(* Schneider Machine Expert - Basic project es3_4pompe_3max_4soglie_misura_livello_con_alternanza_semplice_a_livello_minimo, file version 3.0.0.0 *)
(* ProjectInformations: Name=New project *)

HARDWARE
  Cpu 0: TM221C40R
  ModuleExtensionObject 0: TM3AI8/G
  EthernetConfiguration: NetworkName=M221, IpAllocationMode=FixedAddress, IpAddress=0.0.0.0, SubnetMask=0.0.0.0
  SerialLineConfiguration: Baud=Baud19200, Parity=ParityEven, DataBits=DataBits8, StopBits=StopBits1, PhysicalMedium=PhysicalMediumRs485, TransmissionMode=TransmissionModeModbusRtu, SlaveId=1, Addressing=SlaveAddressing
  MastTask: UsePeriodScanMode=false, PeriodScan=100
  FastTask: Period=255
  CpuBehavior: StartingMode=StartAsPreviousState, AutoSaveRamOnEeprom=true, WatchdogPeriod=250

SYMBOLS  (address, symbol, comment, settings)
  %M0       P1_USABILE
  %M1       P2_USABILE
  %M2       SOTTO_SOGLIA_MIN  "Il livello acqua è passato sotto la soglia minima?"
  %M3       SOPRA_SOGLIA_MAX1  "Il livello acqua è passato sopra la soglia 1 massima?"
  %M4       SOPRA_SOGLIA_MAX2  "Il livello acqua è passato sopra la soglia 2 massima?"
  %M5       PASSATO_SOGLIA_MAX3
  %M6       P1_COMANDATA
  %M7       P2_COMANDATA
  %M8       P3_USABILE
  %M9       P4_USABILE
  %M10      P3_COMANDATA
  %M11      P4_COMANDATA
  %M12      SOPRA_SOGLIA_MAX3  "Il livello acqua è passato sopra la soglia 3 massima?"
  %M13      PASSATO_SOGLIA_MAX2
  %M14      PASSATO_SOGLIA_MAX1
  %MW0      LVL_PERC  "Livello acqua percentuale."
  %MW1      NUM_POMPE_DA_COMANDARE
  %MW2      NUM_POMPE_COMANDATE
  %MD1      LVL_CALC_TMP
  %KD0      MIN_SCALA_GREZZO  [Value=1310724000]
  %KD1      MAX_SCALA_GREZZO  [Value=20000]
  %I0.0     P1_AUTO
  %I0.1     P1_MOTO
  %I0.2     P1_ANOMALIA
  %I0.3     P2_AUTO
  %I0.4     P2_MOTO
  %I0.5     P2_ANOMALIA
  %I0.6     P3_AUTO
  %I0.7     P3_MOTO
  %I0.8     P3_ANOMALIA
  %I0.9     P4_AUTO
  %I0.10    P4_MOTO
  %I0.11    P4_ANOMALIA
  %Q0.0     P1_CMD
  %Q0.1     P2_CMD
  %Q0.2     P3_CMD
  %Q0.3     P4_CMD
  %IW1.0    LVL_INPUT_GREZZO  [Type=Type_4_20mA, Scope=Scope_Customized, Minimum=4000, Maximum=20000]
  %IW1.1    SOGLIA_MIN_PERC  [Type=Type_0_10V, Scope=Scope_Customized, Minimum=0, Maximum=100]
  %IW1.2    SOGLIA_MAX1_PERC  [Type=Type_0_10V, Scope=Scope_Customized, Minimum=0, Maximum=100]
  %IW1.3    SOGLIA_MAX2_PERC  [Type=Type_0_10V, Scope=Scope_Customized, Minimum=0, Maximum=100]
  %IW1.4    SOGLIA_MAX3_PERC  [Type=Type_0_10V, Scope=Scope_Customized, Minimum=0, Maximum=100]

POU Main
  (* SectionNumber=1 *)

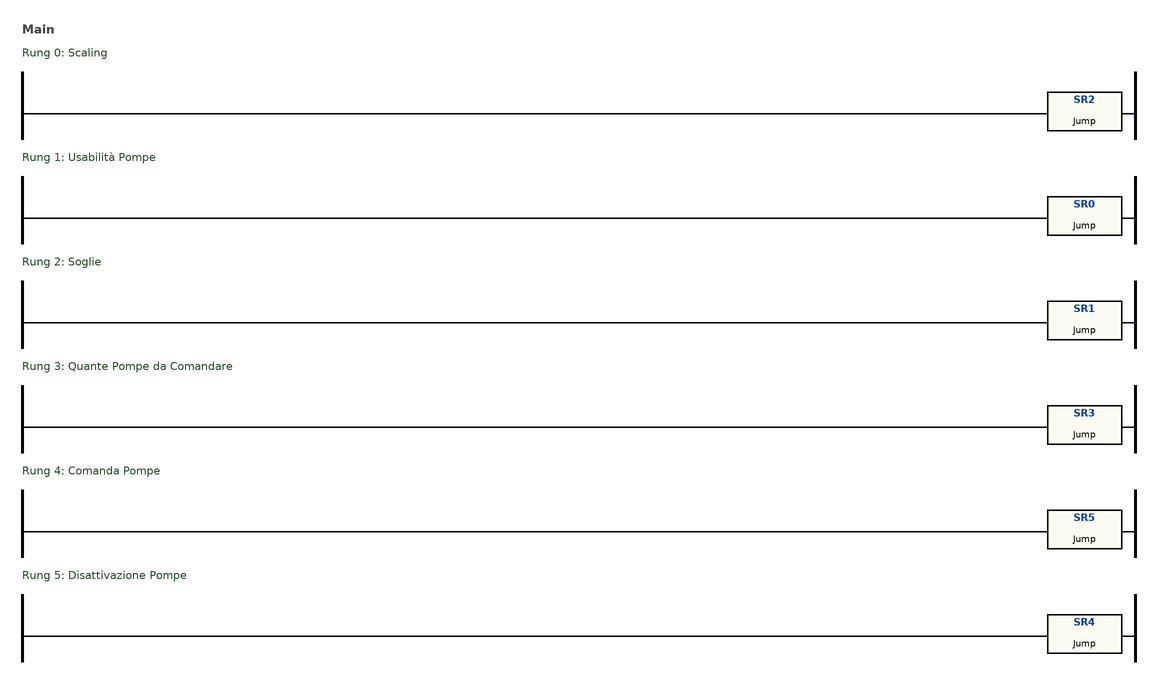

// Rung 0: Scaling
  LD 1
  SR2
  // as ST:
  //   SR2();

// Rung 1: Usabilità Pompe
  LD 1
  SR0
  // as ST:
  //   SR0();

// Rung 2: Soglie
  LD 1
  SR1
  // as ST:
  //   SR1();

// Rung 3: Quante Pompe da Comandare
  LD 1
  SR3
  // as ST:
  //   SR3();

// Rung 4: Comanda Pompe
  LD 1
  SR5
  // as ST:
  //   SR5();

// Rung 5: Disattivazione Pompe
  LD 1
  SR4
  // as ST:
  //   SR4();

Subroutine Usabilità Pompe
  (* SectionNumber=2, Number=0 *)

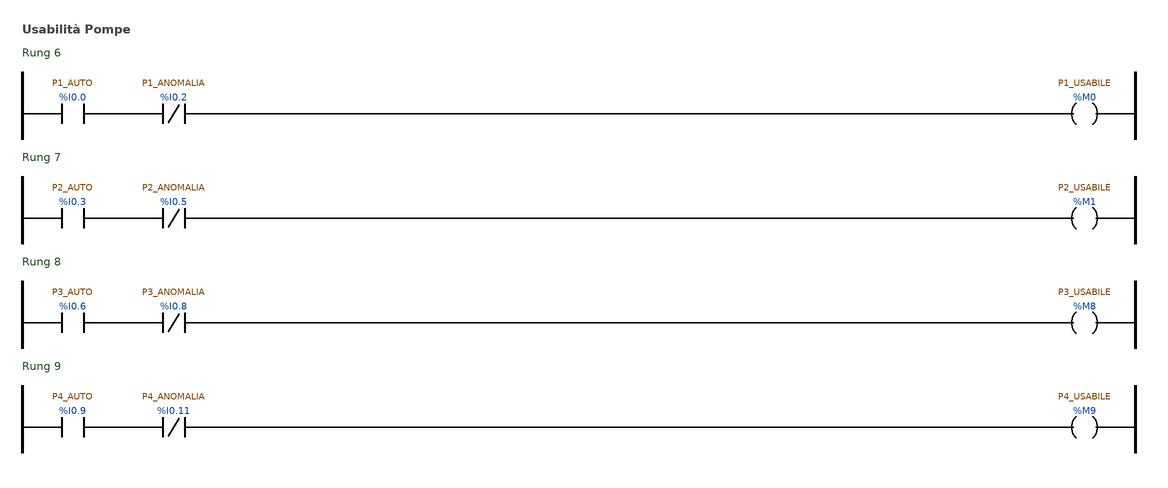

// Rung 6
  LD %I0.0                (* P1_AUTO *)
  ANDN %I0.2              (* P1_ANOMALIA *)
  ST %M0                  (* P1_USABILE *)
  // as ST:
  //   P1_USABILE := P1_AUTO AND NOT P1_ANOMALIA;

// Rung 7
  LD %I0.3                (* P2_AUTO *)
  ANDN %I0.5              (* P2_ANOMALIA *)
  ST %M1                  (* P2_USABILE *)
  // as ST:
  //   P2_USABILE := P2_AUTO AND NOT P2_ANOMALIA;

// Rung 8
  LD %I0.6                (* P3_AUTO *)
  ANDN %I0.8              (* P3_ANOMALIA *)
  ST %M8                  (* P3_USABILE *)
  // as ST:
  //   P3_USABILE := P3_AUTO AND NOT P3_ANOMALIA;

// Rung 9
  LD %I0.9                (* P4_AUTO *)
  ANDN %I0.11             (* P4_ANOMALIA *)
  ST %M9                  (* P4_USABILE *)
  // as ST:
  //   P4_USABILE := P4_AUTO AND NOT P4_ANOMALIA;

Subroutine Soglie
  (* SectionNumber=3, Number=1 *)

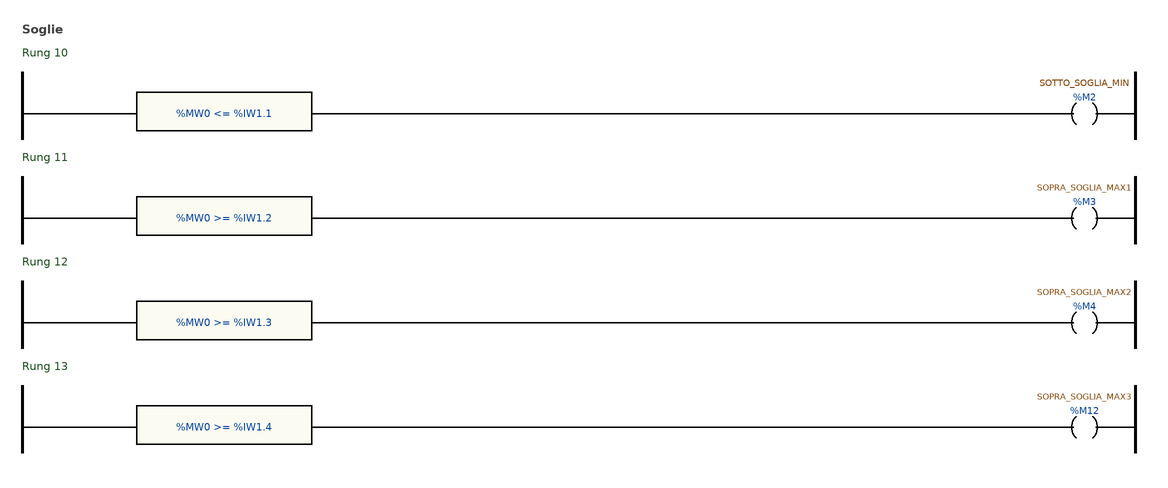

// Rung 10
  LD [ %MW0 <= %IW1.1 ]   (* LVL_PERC, SOGLIA_MIN_PERC *)
  ST %M2                  (* SOTTO_SOGLIA_MIN *)
  // as ST:
  //   SOTTO_SOGLIA_MIN := LVL_PERC <= SOGLIA_MIN_PERC;

// Rung 11
  LD [ %MW0 >= %IW1.2 ]   (* LVL_PERC, SOGLIA_MAX1_PERC *)
  ST %M3                  (* SOPRA_SOGLIA_MAX1 *)
  // as ST:
  //   SOPRA_SOGLIA_MAX1 := LVL_PERC >= SOGLIA_MAX1_PERC;

// Rung 12
  LD [ %MW0 >= %IW1.3 ]   (* LVL_PERC, SOGLIA_MAX2_PERC *)
  ST %M4                  (* SOPRA_SOGLIA_MAX2 *)
  // as ST:
  //   SOPRA_SOGLIA_MAX2 := LVL_PERC >= SOGLIA_MAX2_PERC;

// Rung 13
  LD [ %MW0 >= %IW1.4 ]   (* LVL_PERC, SOGLIA_MAX3_PERC *)
  ST %M12                 (* SOPRA_SOGLIA_MAX3 *)
  // as ST:
  //   SOPRA_SOGLIA_MAX3 := LVL_PERC >= SOGLIA_MAX3_PERC;

Subroutine Scaling
  (* SectionNumber=4, Number=2 *)

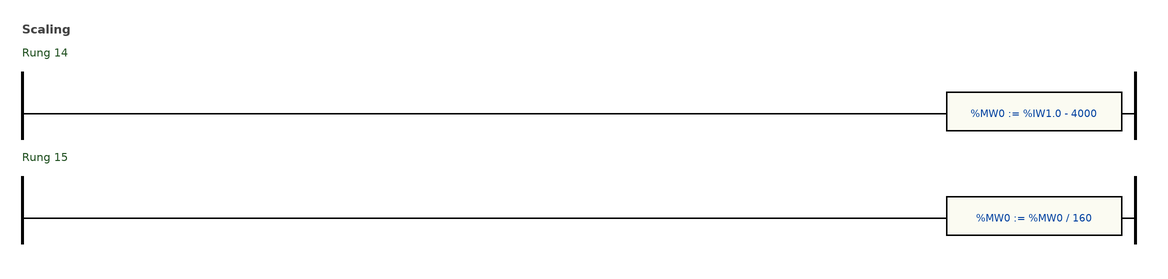

// Rung 14
  LD 1
  [ %MW0 := %IW1.0 - 4000 ](* LVL_PERC, LVL_INPUT_GREZZO *)
  // as ST:
  //   LVL_PERC := LVL_INPUT_GREZZO - 4000;

// Rung 15
  LD 1
  [ %MW0 := %MW0 / 160 ]  (* LVL_PERC, LVL_PERC *)
  // as ST:
  //   LVL_PERC := LVL_PERC / 160;

Subroutine Quante Pompe da Comandare
  (* SectionNumber=5, Number=3 *)

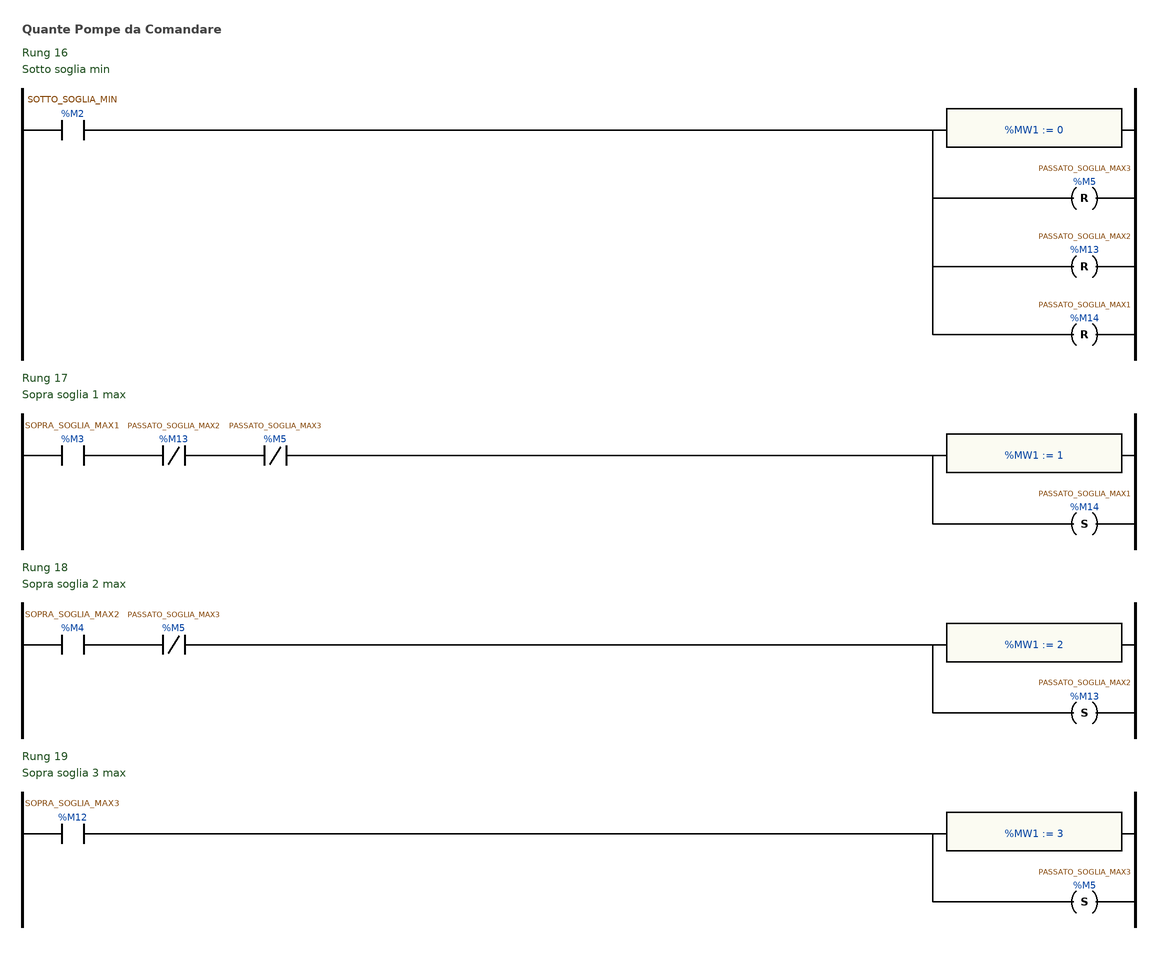

// Rung 16
// Sotto soglia min
  LD %M2                  (* SOTTO_SOGLIA_MIN *)
  [ %MW1 := 0 ]           (* NUM_POMPE_DA_COMANDARE *)
  R %M5                   (* PASSATO_SOGLIA_MAX3 *)
  R %M13                  (* PASSATO_SOGLIA_MAX2 *)
  R %M14                  (* PASSATO_SOGLIA_MAX1 *)
  // as ST:
  //   IF SOTTO_SOGLIA_MIN THEN NUM_POMPE_DA_COMANDARE := 0; END_IF;
  //   IF SOTTO_SOGLIA_MIN THEN PASSATO_SOGLIA_MAX3 := FALSE; END_IF;
  //   IF SOTTO_SOGLIA_MIN THEN PASSATO_SOGLIA_MAX2 := FALSE; END_IF;
  //   IF SOTTO_SOGLIA_MIN THEN PASSATO_SOGLIA_MAX1 := FALSE; END_IF;

// Rung 17
// Sopra soglia 1 max
  LD %M3                  (* SOPRA_SOGLIA_MAX1 *)
  ANDN %M13               (* PASSATO_SOGLIA_MAX2 *)
  ANDN %M5                (* PASSATO_SOGLIA_MAX3 *)
  [ %MW1 := 1 ]           (* NUM_POMPE_DA_COMANDARE *)
  S %M14                  (* PASSATO_SOGLIA_MAX1 *)
  // as ST:
  //   IF SOPRA_SOGLIA_MAX1 AND NOT PASSATO_SOGLIA_MAX2 AND NOT PASSATO_SOGLIA_MAX3 THEN NUM_POMPE_DA_COMANDARE := 1; END_IF;
  //   IF SOPRA_SOGLIA_MAX1 AND NOT PASSATO_SOGLIA_MAX2 AND NOT PASSATO_SOGLIA_MAX3 THEN PASSATO_SOGLIA_MAX1 := TRUE; END_IF;

// Rung 18
// Sopra soglia 2 max
  LD %M4                  (* SOPRA_SOGLIA_MAX2 *)
  ANDN %M5                (* PASSATO_SOGLIA_MAX3 *)
  [ %MW1 := 2 ]           (* NUM_POMPE_DA_COMANDARE *)
  S %M13                  (* PASSATO_SOGLIA_MAX2 *)
  // as ST:
  //   IF SOPRA_SOGLIA_MAX2 AND NOT PASSATO_SOGLIA_MAX3 THEN NUM_POMPE_DA_COMANDARE := 2; END_IF;
  //   IF SOPRA_SOGLIA_MAX2 AND NOT PASSATO_SOGLIA_MAX3 THEN PASSATO_SOGLIA_MAX2 := TRUE; END_IF;

// Rung 19
// Sopra soglia 3 max
  LD %M12                 (* SOPRA_SOGLIA_MAX3 *)
  [ %MW1 := 3 ]           (* NUM_POMPE_DA_COMANDARE *)
  S %M5                   (* PASSATO_SOGLIA_MAX3 *)
  // as ST:
  //   IF SOPRA_SOGLIA_MAX3 THEN NUM_POMPE_DA_COMANDARE := 3; END_IF;
  //   IF SOPRA_SOGLIA_MAX3 THEN PASSATO_SOGLIA_MAX3 := TRUE; END_IF;

Subroutine Disattivazione Pompe
  (* SectionNumber=6, Number=4 *)

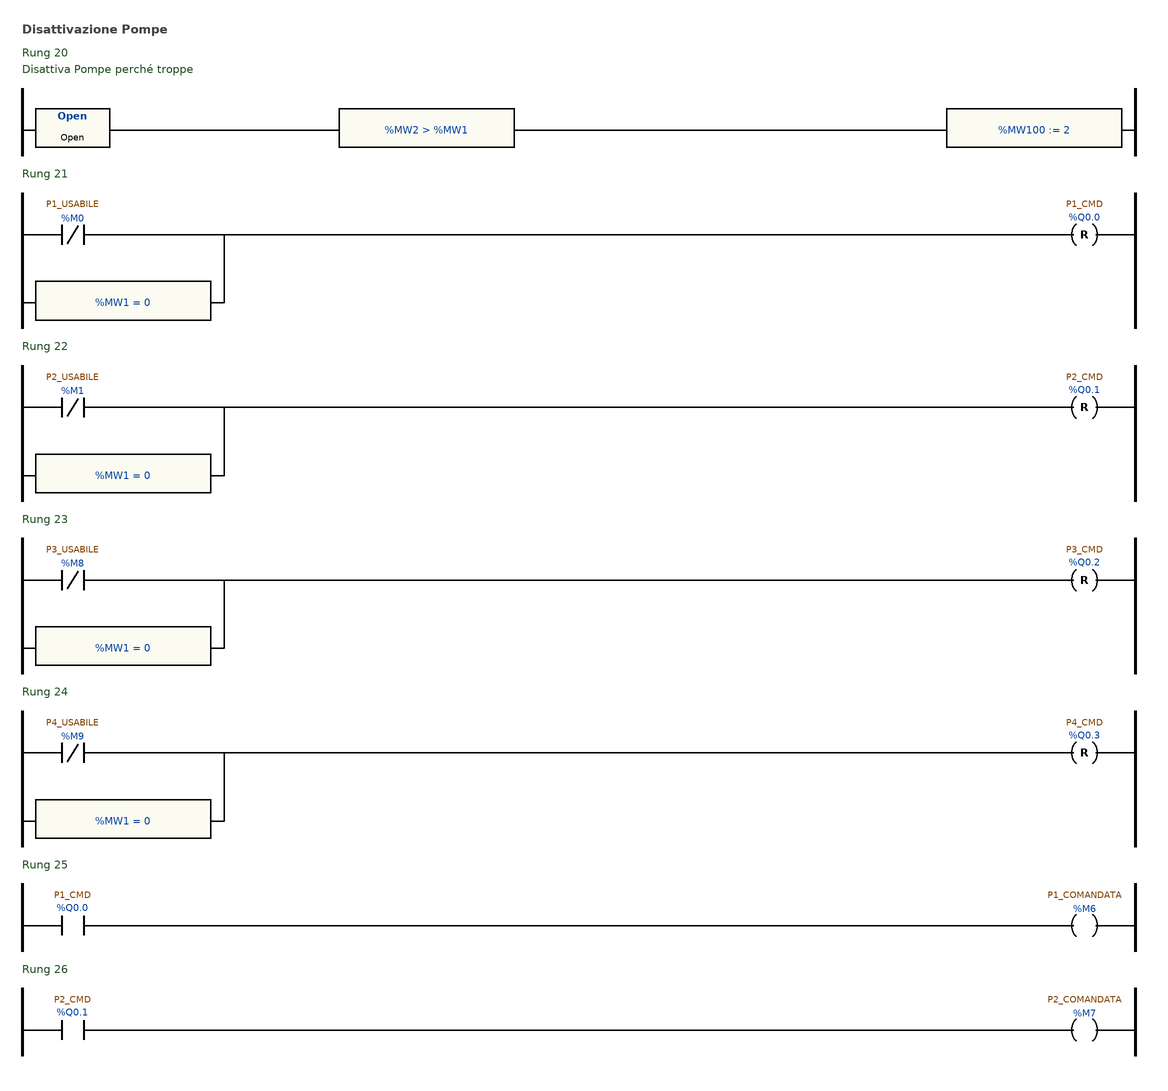

// Rung 20
// Disattiva Pompe perché troppe
  LD 0
  AND [ %MW2 > %MW1 ]     (* NUM_POMPE_COMANDATE, NUM_POMPE_DA_COMANDARE *)
  [ %MW100 := 2 ]
  // as ST:
  //   IF FALSE AND NUM_POMPE_COMANDATE > NUM_POMPE_DA_COMANDARE THEN %MW100 := 2; END_IF;

// Rung 21
  LDN %M0                 (* P1_USABILE *)
  OR [ %MW1 = 0 ]         (* NUM_POMPE_DA_COMANDARE *)
  R %Q0.0                 (* P1_CMD *)
  // as ST:
  //   IF NOT P1_USABILE OR NUM_POMPE_DA_COMANDARE = 0 THEN P1_CMD := FALSE; END_IF;

// Rung 22
  LDN %M1                 (* P2_USABILE *)
  OR [ %MW1 = 0 ]         (* NUM_POMPE_DA_COMANDARE *)
  R %Q0.1                 (* P2_CMD *)
  // as ST:
  //   IF NOT P2_USABILE OR NUM_POMPE_DA_COMANDARE = 0 THEN P2_CMD := FALSE; END_IF;

// Rung 23
  LDN %M8                 (* P3_USABILE *)
  OR [ %MW1 = 0 ]         (* NUM_POMPE_DA_COMANDARE *)
  R %Q0.2                 (* P3_CMD *)
  // as ST:
  //   IF NOT P3_USABILE OR NUM_POMPE_DA_COMANDARE = 0 THEN P3_CMD := FALSE; END_IF;

// Rung 24
  LDN %M9                 (* P4_USABILE *)
  OR [ %MW1 = 0 ]         (* NUM_POMPE_DA_COMANDARE *)
  R %Q0.3                 (* P4_CMD *)
  // as ST:
  //   IF NOT P4_USABILE OR NUM_POMPE_DA_COMANDARE = 0 THEN P4_CMD := FALSE; END_IF;

// Rung 25
  LD %Q0.0                (* P1_CMD *)
  ST %M6                  (* P1_COMANDATA *)
  // as ST:
  //   P1_COMANDATA := P1_CMD;

// Rung 26
  LD %Q0.1                (* P2_CMD *)
  ST %M7                  (* P2_COMANDATA *)
  // as ST:
  //   P2_COMANDATA := P2_CMD;

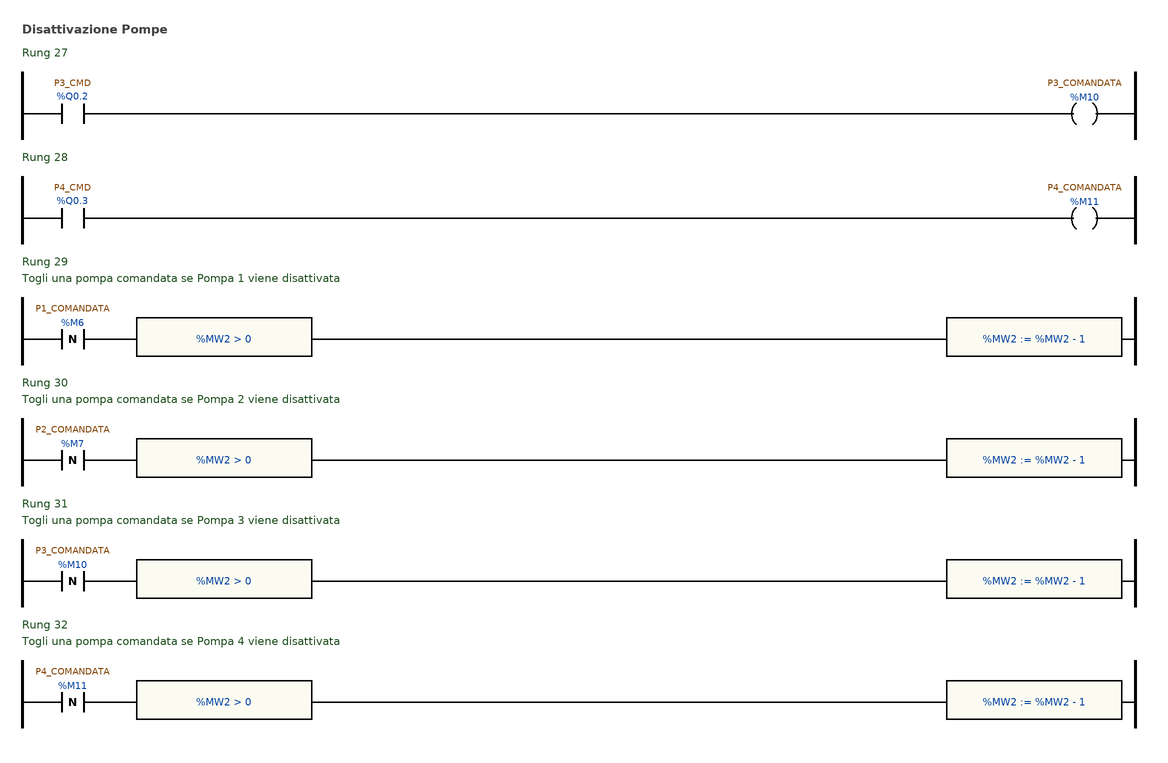

// Rung 27
  LD %Q0.2                (* P3_CMD *)
  ST %M10                 (* P3_COMANDATA *)
  // as ST:
  //   P3_COMANDATA := P3_CMD;

// Rung 28
  LD %Q0.3                (* P4_CMD *)
  ST %M11                 (* P4_COMANDATA *)
  // as ST:
  //   P4_COMANDATA := P4_CMD;

// Rung 29
// Togli una pompa comandata se Pompa 1 viene disattivata
  LDF %M6                 (* P1_COMANDATA *)
  AND [ %MW2 > 0 ]        (* NUM_POMPE_COMANDATE *)
  [ %MW2 := %MW2 - 1 ]    (* NUM_POMPE_COMANDATE, NUM_POMPE_COMANDATE *)
  // as ST:
  //   IF FALLING(P1_COMANDATA) AND NUM_POMPE_COMANDATE > 0 THEN NUM_POMPE_COMANDATE := NUM_POMPE_COMANDATE - 1; END_IF;

// Rung 30
// Togli una pompa comandata se Pompa 2 viene disattivata
  LDF %M7                 (* P2_COMANDATA *)
  AND [ %MW2 > 0 ]        (* NUM_POMPE_COMANDATE *)
  [ %MW2 := %MW2 - 1 ]    (* NUM_POMPE_COMANDATE, NUM_POMPE_COMANDATE *)
  // as ST:
  //   IF FALLING(P2_COMANDATA) AND NUM_POMPE_COMANDATE > 0 THEN NUM_POMPE_COMANDATE := NUM_POMPE_COMANDATE - 1; END_IF;

// Rung 31
// Togli una pompa comandata se Pompa 3 viene disattivata
  LDF %M10                (* P3_COMANDATA *)
  AND [ %MW2 > 0 ]        (* NUM_POMPE_COMANDATE *)
  [ %MW2 := %MW2 - 1 ]    (* NUM_POMPE_COMANDATE, NUM_POMPE_COMANDATE *)
  // as ST:
  //   IF FALLING(P3_COMANDATA) AND NUM_POMPE_COMANDATE > 0 THEN NUM_POMPE_COMANDATE := NUM_POMPE_COMANDATE - 1; END_IF;

// Rung 32
// Togli una pompa comandata se Pompa 4 viene disattivata
  LDF %M11                (* P4_COMANDATA *)
  AND [ %MW2 > 0 ]        (* NUM_POMPE_COMANDATE *)
  [ %MW2 := %MW2 - 1 ]    (* NUM_POMPE_COMANDATE, NUM_POMPE_COMANDATE *)
  // as ST:
  //   IF FALLING(P4_COMANDATA) AND NUM_POMPE_COMANDATE > 0 THEN NUM_POMPE_COMANDATE := NUM_POMPE_COMANDATE - 1; END_IF;

Subroutine Comanda Pompe
  (* SectionNumber=7, Number=5 *)

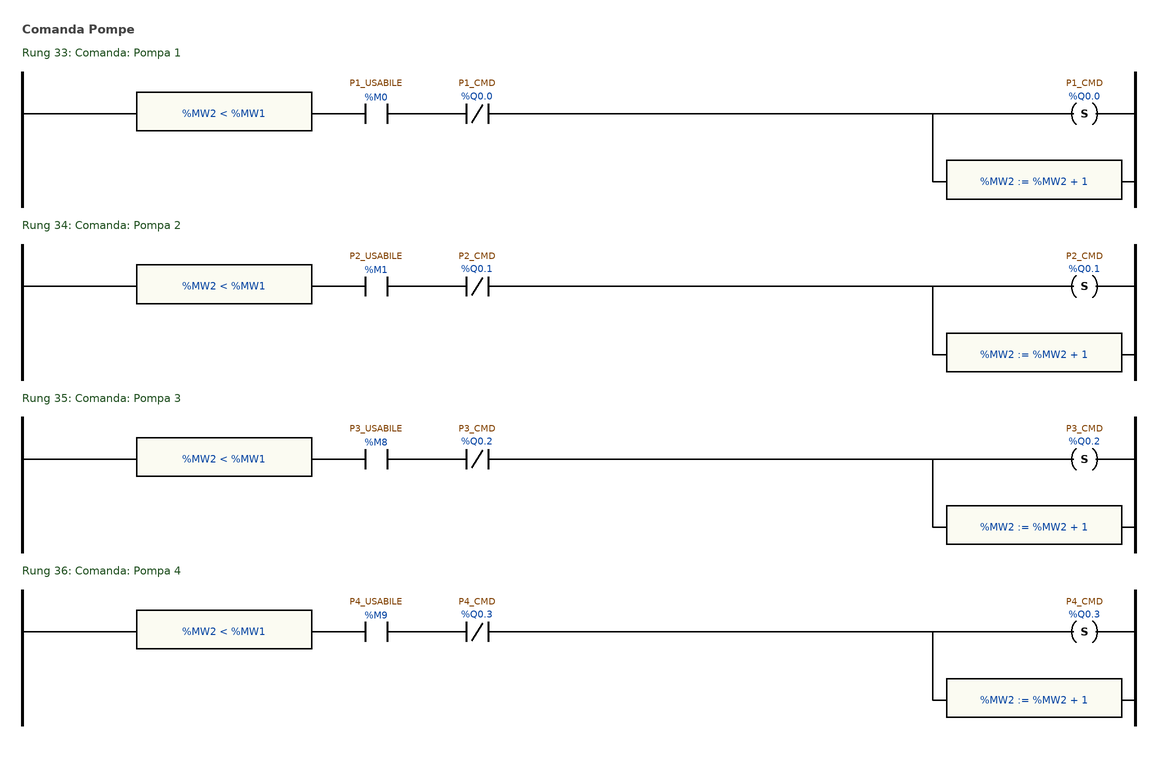

// Rung 33: Comanda: Pompa 1
  LD [ %MW2 < %MW1 ]      (* NUM_POMPE_COMANDATE, NUM_POMPE_DA_COMANDARE *)
  AND %M0                 (* P1_USABILE *)
  ANDN %Q0.0              (* P1_CMD *)
  S %Q0.0                 (* P1_CMD *)
  [ %MW2 := %MW2 + 1 ]    (* NUM_POMPE_COMANDATE, NUM_POMPE_COMANDATE *)
  // as ST:
  //   _t1 := NUM_POMPE_COMANDATE < NUM_POMPE_DA_COMANDARE AND P1_USABILE AND NOT P1_CMD;
  //   IF _t1 THEN P1_CMD := TRUE; END_IF;
  //   IF _t1 THEN NUM_POMPE_COMANDATE := NUM_POMPE_COMANDATE + 1; END_IF;

// Rung 34: Comanda: Pompa 2
  LD [ %MW2 < %MW1 ]      (* NUM_POMPE_COMANDATE, NUM_POMPE_DA_COMANDARE *)
  AND %M1                 (* P2_USABILE *)
  ANDN %Q0.1              (* P2_CMD *)
  S %Q0.1                 (* P2_CMD *)
  [ %MW2 := %MW2 + 1 ]    (* NUM_POMPE_COMANDATE, NUM_POMPE_COMANDATE *)
  // as ST:
  //   _t1 := NUM_POMPE_COMANDATE < NUM_POMPE_DA_COMANDARE AND P2_USABILE AND NOT P2_CMD;
  //   IF _t1 THEN P2_CMD := TRUE; END_IF;
  //   IF _t1 THEN NUM_POMPE_COMANDATE := NUM_POMPE_COMANDATE + 1; END_IF;

// Rung 35: Comanda: Pompa 3
  LD [ %MW2 < %MW1 ]      (* NUM_POMPE_COMANDATE, NUM_POMPE_DA_COMANDARE *)
  AND %M8                 (* P3_USABILE *)
  ANDN %Q0.2              (* P3_CMD *)
  S %Q0.2                 (* P3_CMD *)
  [ %MW2 := %MW2 + 1 ]    (* NUM_POMPE_COMANDATE, NUM_POMPE_COMANDATE *)
  // as ST:
  //   _t1 := NUM_POMPE_COMANDATE < NUM_POMPE_DA_COMANDARE AND P3_USABILE AND NOT P3_CMD;
  //   IF _t1 THEN P3_CMD := TRUE; END_IF;
  //   IF _t1 THEN NUM_POMPE_COMANDATE := NUM_POMPE_COMANDATE + 1; END_IF;

// Rung 36: Comanda: Pompa 4
  LD [ %MW2 < %MW1 ]      (* NUM_POMPE_COMANDATE, NUM_POMPE_DA_COMANDARE *)
  AND %M9                 (* P4_USABILE *)
  ANDN %Q0.3              (* P4_CMD *)
  S %Q0.3                 (* P4_CMD *)
  [ %MW2 := %MW2 + 1 ]    (* NUM_POMPE_COMANDATE, NUM_POMPE_COMANDATE *)
  // as ST:
  //   _t1 := NUM_POMPE_COMANDATE < NUM_POMPE_DA_COMANDARE AND P4_USABILE AND NOT P4_CMD;
  //   IF _t1 THEN P4_CMD := TRUE; END_IF;
  //   IF _t1 THEN NUM_POMPE_COMANDATE := NUM_POMPE_COMANDATE + 1; END_IF;
